FUNCTION_BLOCK INTERNAL ABSTRACT FB_FieldCodec IMPLEMENTS I_FieldCodec
VAR_INPUT
END_VAR
VAR_OUTPUT
END_VAR
VAR	
	nTagField				: UDINT;
	nEndTagField			: UDINT;
    ipMessageField          : I_Message;
END_VAR

{attribute 'no-analysis'}
METHOD ABSTRACT CalculatePackedDataSize : HRESULT
VAR_INPUT
	anyFirstElem	: T_Any;
	(* items to write*)
	nLength	: UDINT;
END_VAR
VAR_OUTPUT
	nPackedDataSize	: UDINT;
END_VAR
END_METHOD

{warning 'Add property implementation'}
(* Gets the end tag of the codec or 0 if there is no end tag*)
PROPERTY EndTag : UDINT
GET
EndTag := THIS^.nEndTagField;
END_GET
SET
THIS^.nEndTagField := EndTag;
END_SET
END_PROPERTY

//FB_Init is always available implicitly and it is used primarily for initialization.
//The return value is not evaluated. For a specific influence, you can also declare the
//methods explicitly and provide additional code there with the standard initialization
//code. You can evaluate the return value.
METHOD FB_Init: BOOL
VAR_INPUT
    bInitRetains: BOOL; // TRUE: the retain variables are initialized (reset warm / reset cold)
    bInCopyCode: BOOL;  // TRUE: the instance will be copied to the copy code afterward (online change)
	nTag : UDINT;
END_VAR
THIS^.nTagField := nTag;
END_METHOD

// The I_Message for this FieldCodec
PROPERTY ipMessage : I_Message
GET
ipMessage := THIS^.ipMessageField;
END_GET
SET
THIS^.ipMessageField := ipMessage;
END_SET
END_PROPERTY

{attribute 'no-analysis'}
METHOD ABSTRACT IsPackedRepeatedField : BOOL
VAR_INPUT
	nTag	: UDINT;
END_VAR
END_METHOD

{warning 'Add property implementation'}
(* Gets the tag of the codec.*)
PROPERTY Tag : UDINT
GET
Tag := THIS^.nTagField;
END_GET
SET
THIS^.nTagField := Tag;
END_SET
END_PROPERTY

{attribute 'no-analysis'}
METHOD ABSTRACT ValueReader : HRESULT
VAR_IN_OUT
	stCtx	: ST_ParseContext;
END_VAR
VAR_OUTPUT
	anyOut	: T_Any;
END_VAR
END_METHOD

{attribute 'no-analysis'}
METHOD ABSTRACT ValueWriter : HRESULT
VAR_IN_OUT
	stCtx	: ST_WriteContext;
END_VAR
VAR_INPUT
	anyIn	: T_ANY;
END_VAR
END_METHOD

END_FUNCTION_BLOCK

(* stored: Version 1.1.0.1
   POU FB_FieldCodec: Id {6f6b06a5-a8a9-4112-8bc8-645fce5ed92c}, SpecialFunc None
   Method CalculatePackedDataSize: Id {eba1a773-8167-4bdb-aaa6-213f64cdea6c}
   Property EndTag: Id {7644fe42-2647-46e2-b811-2142c17e2a15}
   Get Get: Id {b15dc5fa-8a08-4a7d-a223-d7a42fa20cf7}
   Set Set: Id {97706bdf-9008-4e69-a7fa-e305ca386419}
   Method FB_Init: Id {16d4c543-9c15-4ce2-a3cc-687ffea975c7}
   Property ipMessage: Id {87ab2de9-fddd-4bb7-8ba5-30028794b2ca}
   Get Get: Id {a7b6b2dd-0fbc-4fb4-9524-7e9116364345}
   Set Set: Id {912eb063-e4b5-41b4-a5cc-a2f9442b3648}
   Method IsPackedRepeatedField: Id {526d0a88-3154-4737-9e80-8d4a872f9c83}
   Property Tag: Id {ca6415b5-e709-4327-aee2-f3dc4fe3c7b1}
   Get Get: Id {5d751c95-c1a2-4d05-b6fb-522a0897af45}
   Set Set: Id {3401ac34-7798-4468-9426-a31d0ce1ab1c}
   Method ValueReader: Id {94e8bf03-4b1f-459b-9d24-d4a8f124423a}
   Method ValueWriter: Id {247f3b40-a101-431e-aac2-ae10ff555ab4} *)
